FUNCTION F_CheckAxisLES : BOOL
VAR_INPUT
    stMotionStage: ST_MotionStage;
    fQueryValue: LREAL;
END_VAR
VAR
END_VAR


F_CheckAxisLES := F_CheckAxis(stMotionStage, 0, fQueryValue);

END_FUNCTION

(* stored: Version 1.1.0.1
   POU F_CheckAxisLES: Id {0c65dbf2-5903-404f-946d-2e0fda97e3ea}, SpecialFunc None *)
